PROGRAM MAIN
VAR
	
fb_solvexy:FB_SOLVEXY;
	error AT %Q*: BOOL;

END_VAR

GVL.blink := NOT(GVL.blink);

fb_solvexy.x:=GVL.Xc;
fb_solvexy.y:=GVL.Yc;
fb_solvexy();
GVL.d1 :=fb_solvexy.d1;
GVL.d2 :=fb_solvexy.d2;
error := fb_solvexy.error;
GVL.alfa1:=180/GVL.Pi*fb_solvexy.alfa1;
GVL.beta1:=180/GVL.Pi*fb_solvexy.beta1;
GVL.alfa2:=180/GVL.Pi*fb_solvexy.alfa2;
GVL.beta2:=180/GVL.Pi*fb_solvexy.beta2;
GVL.alfa:=180/GVL.Pi*fb_solvexy.alfa;
GVL.beta:=180/GVL.Pi*fb_solvexy.beta;

END_PROGRAM

(* stored: Version 1.1.0.1, ProductVersion 3.1.4024.4
   POU MAIN: Id {d89af4a1-5c9c-4631-9fc2-66e77163c97b}, SpecialFunc None *)
